FUNCTION F_DeviceState_To_DeviceStateExt : ST_DeviceStateExt
VAR_INPUT
    stDeviceState    :    ST_DeviceState;
    xValid    :    BOOL;
END_VAR
VAR
END_VAR

F_DeviceState_To_DeviceStateExt.nStateRef := stDeviceState.nStateRef;
F_DeviceState_To_DeviceStateExt.rPosition    :=    stDeviceState.rPosition;
F_DeviceState_To_DeviceStateExt.rTolerance    :=    stDeviceState.rTolerance;
F_DeviceState_To_DeviceStateExt.sStateName    := stDeviceState.sStateName;
F_DeviceState_To_DeviceStateExt.stReqBeamParam    := stDeviceState.stReqBeamParam;
F_DeviceState_To_DeviceStateExt.xValid := xValid;

END_FUNCTION

(* stored: Version 1.1.0.1
   POU F_DeviceState_To_DeviceStateExt: Id {647f5b20-e140-4a4a-b23d-0cce310441de}, SpecialFunc None *)
